(* PLC project SootBlower, Unknown Unnamed 1 *)
(* stored: creationDateTime 2024-10-02T21:08:56, modificationDateTime 2024-10-04T16:07:09 *)

PROGRAM program0
  VAR
    Start AT %IX0.0 : BOOL;
    Stop AT %IX0.1 : BOOL;
    Alarm AT %IX0.2 : BOOL;
    Green AT %QX0.0 : BOOL;
    Red AT %QX0.1 : BOOL;
    Motor AT %QX0.2 : BOOL;
    Buzzer AT %QX0.3 : BOOL;
    Blink_Pulse AT %QX0.4 : BOOL;
    Running AT %QX0.5 : BOOL;
  END_VAR
  VAR
    TON0 : TON;
    TOF0 : TOF;
  END_VAR

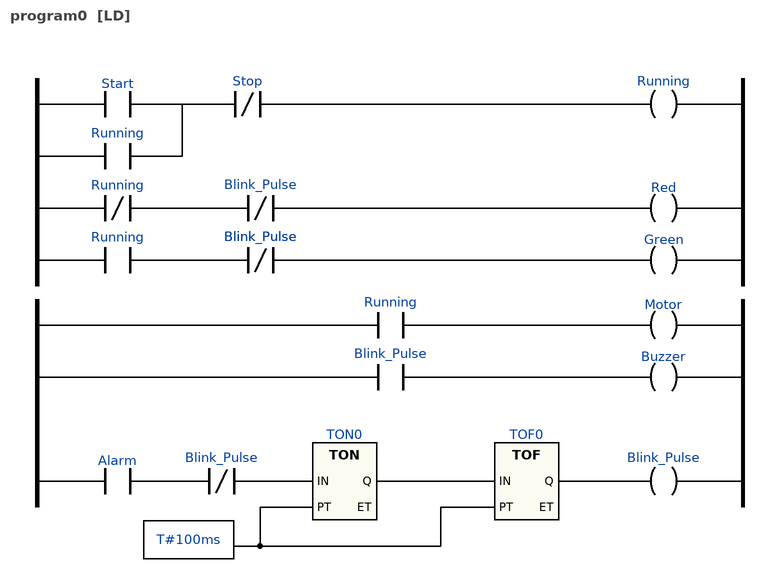
(* LD diagram, written out as Structured Text *)
Running := (Start OR Running) AND NOT Stop;
Red := NOT Running AND NOT Blink_Pulse;
Green := Running AND NOT Blink_Pulse;
TON0(IN := Alarm AND NOT Blink_Pulse, PT := T#100ms);
TOF0(IN := TON0.Q, PT := T#100ms);
Blink_Pulse := TOF0.Q;
Motor := Running;
Buzzer := Blink_Pulse;
(* drawn but not wired to any output: Blink_Pulse *)
END_PROGRAM

CONFIGURATION Config0
  RESOURCE Res0 ON PLC
    TASK task0(INTERVAL := T#20ms, PRIORITY := 0);
    PROGRAM instance0 WITH task0 : program0;
  END_RESOURCE
END_CONFIGURATION
